{attribute 'linkalways'} 
{attribute 'no_explicit_call' := 'This FB is a CLASS and must be accessed using methods or properties'}
{attribute 'enable_dynamic_creation'}
FUNCTION_BLOCK _ETcVnClusteringAlgorithm EXTENDS EnumDatatypeBase
VAR
	localData : ETcVnClusteringAlgorithm;
	activeData : REFERENCE TO ETcVnClusteringAlgorithm;
	enumBaseDatatype : _DINT(localData);
END_VAR

METHOD PRIVATE AddLocalEnumeration
VAR_INPUT
	Enumeration : T_MAXSTRING;
	Value : ETcVnClusteringAlgorithm;
END_VAR
AddEnumeration(Enumeration, Value);
END_METHOD

PROPERTY PUBLIC Address : PVOID
GET
Address := ADR(activeData);
END_GET
END_PROPERTY

METHOD PUBLIC ClearReference
VAR_INPUT
END_VAR
activeData REF= localData;
SetBaseDatatypeReference();
END_METHOD

METHOD PUBLIC Clone : I_Datatype
VAR
    pClone : POINTER TO _ETcVnClusteringAlgorithm;
END_VAR
pClone := __NEW(_ETcVnClusteringAlgorithm(InitialValue := Value));
Clone := pClone^;
END_METHOD

METHOD FB_init : BOOL
VAR_INPUT
	bInitRetains : BOOL; // if TRUE, the retain variables are initialized (warm start / cold start)
	bInCopyCode : BOOL;  // if TRUE, the instance afterwards gets moved into the copy code (online change)
	InitialValue : ETcVnClusteringAlgorithm;
END_VAR
localData := InitialValue;
AddBaseDatatype(enumBaseDatatype);
ClearReference();

AddLocalEnumeration('TCVN_CA_KMEANSPP', ETcVnClusteringAlgorithm.TCVN_CA_KMEANSPP);
AddLocalEnumeration('TCVN_CA_LBG', ETcVnClusteringAlgorithm.TCVN_CA_LBG);
END_METHOD

PROPERTY PUBLIC Identifier : T_MAXSTRING
GET
Identifier := 'ETcVnClusteringAlgorithm';
END_GET
END_PROPERTY

METHOD IsEnumeratorValueEqual : BOOL
VAR_INPUT
	Enumerator : I_KeyValueForwardEnumerator;
END_VAR
VAR
	storedValue : ETcVnClusteringAlgorithm;
END_VAR
IF NOT Enumerator.TryGet(storedValue) THEN
	RETURN;
END_IF

IsEnumeratorValueEqual := storedValue = activeData;
END_METHOD

METHOD PUBLIC MakeReferenceTo
VAR_INPUT
	ReferenceTarget : REFERENCE TO ETcVnCalibrationPatternOrigin;
END_VAR
activeData REF= ReferenceTarget;
SetBaseDatatypeReference();
END_METHOD

METHOD PROTECTED SetBaseDatatypeReference
VAR_INPUT
END_VAR
enumBaseDatatype.MakeReferenceTo(activeData);
END_METHOD

PROPERTY PUBLIC Size : UDINT
GET
Size := SIZEOF(activeData);
END_GET
END_PROPERTY

METHOD TryMakeReferenceTo : BOOL
VAR_INPUT
	Target : I_Datatype;
END_VAR
VAR
	targetAsEnum : I_EnumDatatype;
	pTargetData : POINTER TO ETcVnClusteringAlgorithm;
END_VAR
IF NOT Target.TryResolveAsEnumDatatype(targetAsEnum) THEN
	RETURN;
END_IF

IF targetAsEnum.Identifier <> Identifier THEN
	RETURN;
END_IF

pTargetData := Target.Address;
activeData REF= pTargetData^;
SetBaseDatatypeReference();
TryMakeReferenceTo := TRUE;
END_METHOD

PROPERTY PUBLIC Value : ETcVnClusteringAlgorithm
GET
Value := activeData;
END_GET
SET
activeData := Value;
END_SET
END_PROPERTY

END_FUNCTION_BLOCK

(* stored: Version 1.1.0.1, ProductVersion 3.1.4024.12
   POU _ETcVnClusteringAlgorithm: Id {bd67b116-e437-0faf-250d-6ff45902e4ab}, SpecialFunc None
   Folder Constructor: Id {bd5b8375-9351-043a-2c6f-f3b9b85ef1c8}
   Folder Private: Id {ae307fae-554c-04b5-3536-5963eb3af9f5}
   Folder Protected: Id {35403e5f-05db-0e08-0005-a1e942031190}
   Method AddLocalEnumeration: Id {46bf60e3-8198-04ad-2dce-e6d548ba69b3}
   Property Address: Id {138928c5-b1bd-0aaa-35bc-93d5657d2ddc}
   Get Get: Id {c83d58ec-bfd2-0489-0e80-383f0ed8c26b}
   Method ClearReference: Id {2baf302b-b258-0b98-2e69-663f763c8966}
   Method Clone: Id {ff16f5fa-1326-088d-1199-ad0a0a87c263}
   Method FB_init: Id {091b644c-b59a-0bf7-0275-1f9a10c86022}
   Property Identifier: Id {677ac972-88f9-0393-03c7-78122534570c}
   Get Get: Id {815c7f25-5aaf-079b-36d3-cc3dc083bfb4}
   Method IsEnumeratorValueEqual: Id {8447de0e-756b-0f00-14f1-89ec240ee3c7}
   Method MakeReferenceTo: Id {daddc33c-6236-0858-1f8b-ee9b6e601203}
   Method SetBaseDatatypeReference: Id {500478e6-644d-03cf-0ff6-96ca3fe18911}
   Property Size: Id {204c0d38-5460-067d-119a-35df54641c7d}
   Get Get: Id {3cb1b40d-8d1d-06e4-149d-b9dc2db037cc}
   Method TryMakeReferenceTo: Id {5032dadb-1214-0bce-3e2d-9f1208a9274a}
   Property Value: Id {ac4a3fee-b46e-0986-36ac-e8819625067a}
   Get Get: Id {113b6b9c-9314-0f08-0d3e-56d0633ddd11}
   Set Set: Id {7d62044d-d8e8-0a95-1a01-ebb6d72bcbbf} *)
